(* Logix 5000 project; controller SX_V040001_C001 vendor 1 type 14 code 77 rev 16.23; software revision 16.04; part 12 of 35 *)
(* tags used below, declared in another part *)
   ALL_KINDS : INT[90];
   Basic : INT;
   C_MINUTES : COUNTER;
   C_SECONDS : COUNTER;
   CMD : INT[36];
   DRIVE : INT[32];
   DRIVE_INTERVAL : INT[8];
   EMPTYING : INT[18];
   G_DInput : DINT[3];
   G_DOutput : DINT[3];
   loading : INT[19];
   louvre : INT[11];
   m_alarm_exist : BOOL;
   m_alarm_horn : BOOL;
   m_battery_low : BOOL;
   m_on_off_line : BOOL;
   m_power_up : BOOL;
   PARAMETER : INT[501];
   STATUS_GENERAL : INT[135];
   TEMP : INT[14];
(* MainProgram, continued *)

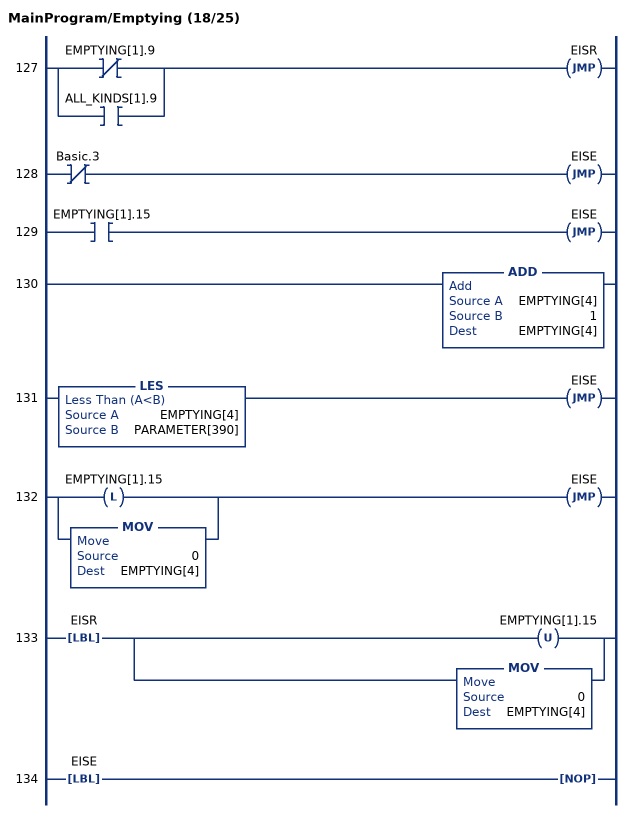
   [picture p256: MainProgram/Emptying rungs 127-134]
   127: [XIO(EMPTYING[1].9) ,XIC(ALL_KINDS[1].9) ]JMP(EISR);
   128: XIO(Basic.3)JMP(EISE);
   129: XIC(EMPTYING[1].15)JMP(EISE);
   130: ADD(EMPTYING[4],1,EMPTYING[4]);
   131: LES(EMPTYING[4],PARAMETER[390])JMP(EISE);
   132: [OTL(EMPTYING[1].15) ,MOV(0,EMPTYING[4]) ]JMP(EISE);
   133: LBL(EISR)[OTU(EMPTYING[1].15) ,MOV(0,EMPTYING[4]) ];
   134: LBL(EISE)NOP();
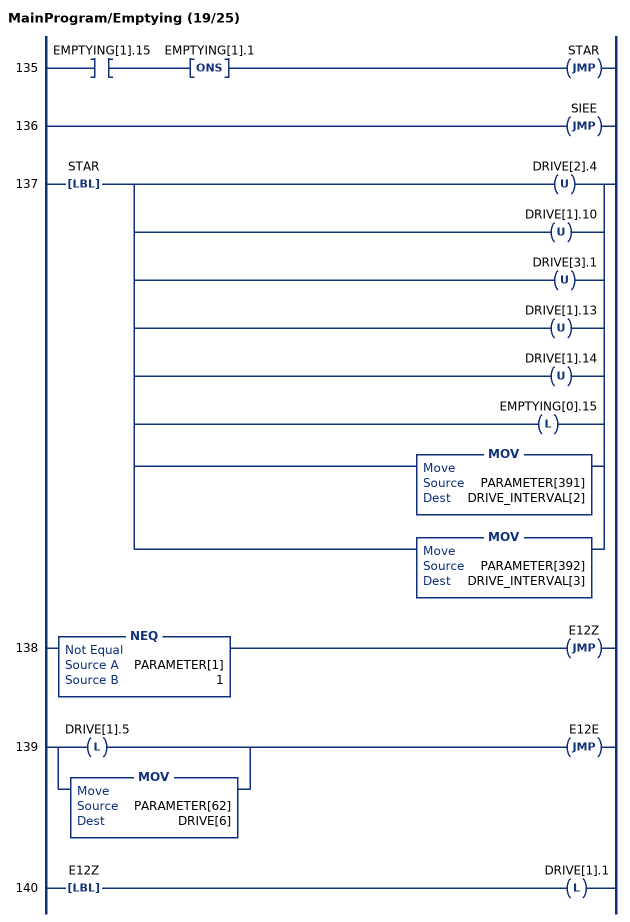
   135: XIC(EMPTYING[1].15)ONS(EMPTYING[1].1)JMP(STAR);
   136: JMP(SIEE);
   137: LBL(STAR)[OTU(DRIVE[2].4) ,OTU(DRIVE[1].10) ,OTU(DRIVE[3].1) ,OTU(DRIVE[1].13) ,OTU(DRIVE[1].14) ,OTL(EMPTYING[0].15) ,MOV(PARAMETER[391],DRIVE_INTERVAL[2]) ,MOV(PARAMETER[392],DRIVE_INTERVAL[3]) ];
   138: NEQ(PARAMETER[1],1)JMP(E12Z);
   139: [OTL(DRIVE[1].5) ,MOV(PARAMETER[62],DRIVE[6]) ]JMP(E12E);
   140: LBL(E12Z)OTL(DRIVE[1].1);
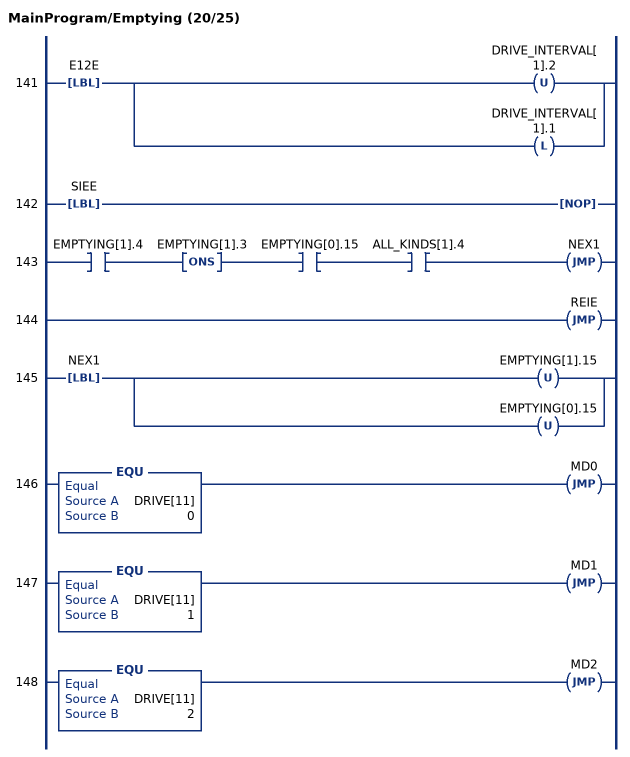
   141: LBL(E12E)[OTU(DRIVE_INTERVAL[1].2) ,OTL(DRIVE_INTERVAL[1].1) ];
   142: LBL(SIEE)NOP();
   143: XIC(EMPTYING[1].4)ONS(EMPTYING[1].3)XIC(EMPTYING[0].15)XIC(ALL_KINDS[1].4)JMP(NEX1);
   144: JMP(REIE);
   145: LBL(NEX1)[OTU(EMPTYING[1].15) ,OTU(EMPTYING[0].15) ];
   146: EQU(DRIVE[11],0)JMP(MD0);
   147: EQU(DRIVE[11],1)JMP(MD1);
   148: EQU(DRIVE[11],2)JMP(MD2);
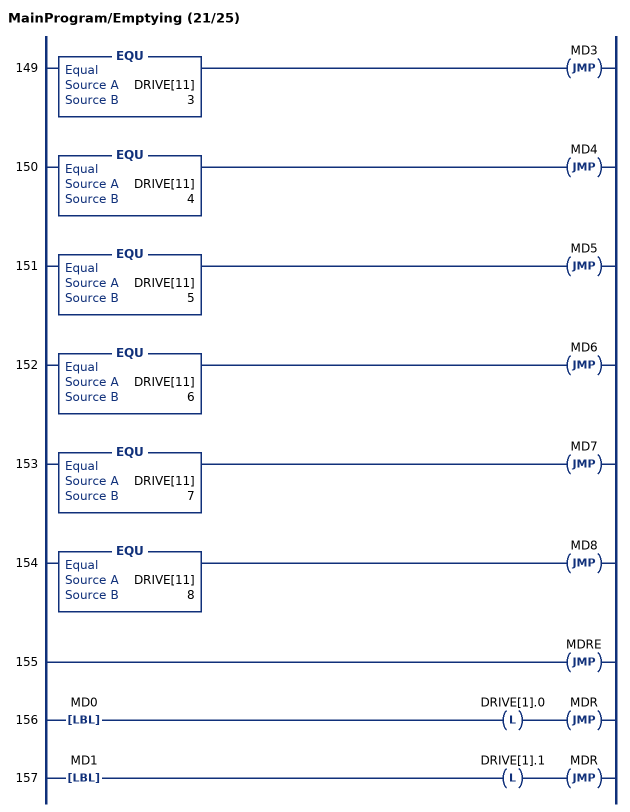
   149: EQU(DRIVE[11],3)JMP(MD3);
   150: EQU(DRIVE[11],4)JMP(MD4);
   151: EQU(DRIVE[11],5)JMP(MD5);
   152: EQU(DRIVE[11],6)JMP(MD6);
   153: EQU(DRIVE[11],7)JMP(MD7);
   154: EQU(DRIVE[11],8)JMP(MD8);
   155: JMP(MDRE);
   156: LBL(MD0)OTL(DRIVE[1].0)JMP(MDR);
   157: LBL(MD1)OTL(DRIVE[1].1)JMP(MDR);
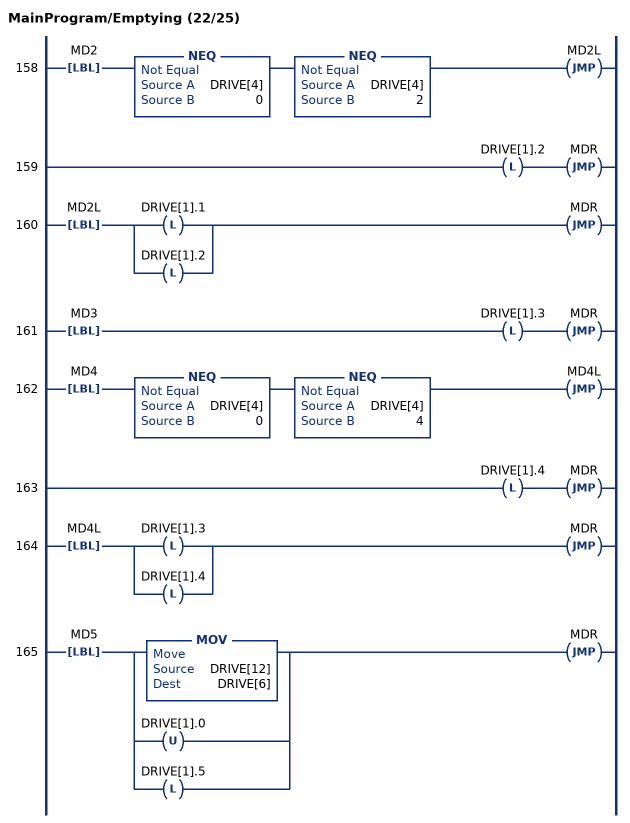
   158: LBL(MD2)NEQ(DRIVE[4],0)NEQ(DRIVE[4],2)JMP(MD2L);
   159: OTL(DRIVE[1].2)JMP(MDR);
   160: LBL(MD2L)[OTL(DRIVE[1].1) ,OTL(DRIVE[1].2) ]JMP(MDR);
   161: LBL(MD3)OTL(DRIVE[1].3)JMP(MDR);
   162: LBL(MD4)NEQ(DRIVE[4],0)NEQ(DRIVE[4],4)JMP(MD4L);
   163: OTL(DRIVE[1].4)JMP(MDR);
   164: LBL(MD4L)[OTL(DRIVE[1].3) ,OTL(DRIVE[1].4) ]JMP(MDR);
   165: LBL(MD5)[MOV(DRIVE[12],DRIVE[6]) ,OTU(DRIVE[1].0) ,OTL(DRIVE[1].5) ]JMP(MDR);
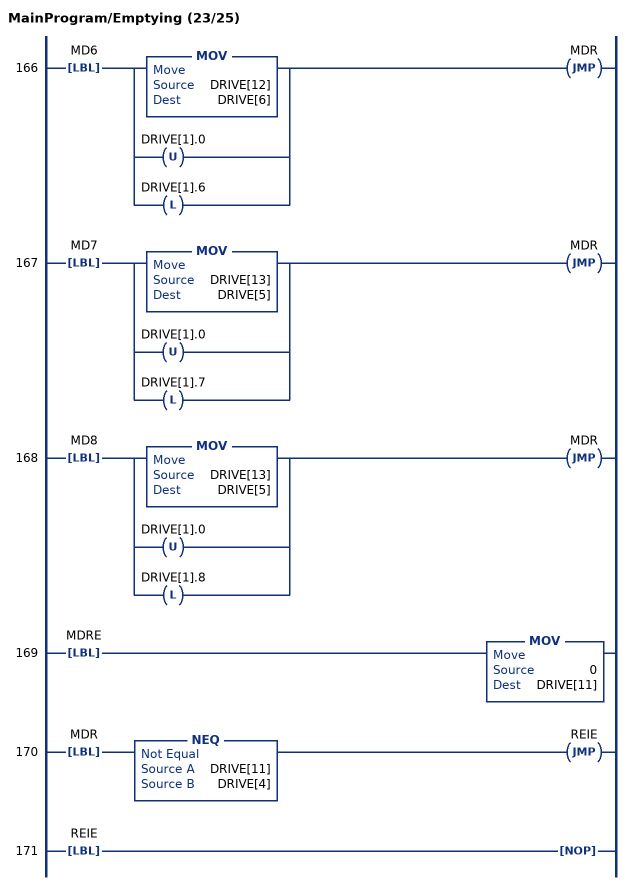
   166: LBL(MD6)[MOV(DRIVE[12],DRIVE[6]) ,OTU(DRIVE[1].0) ,OTL(DRIVE[1].6) ]JMP(MDR);
   167: LBL(MD7)[MOV(DRIVE[13],DRIVE[5]) ,OTU(DRIVE[1].0) ,OTL(DRIVE[1].7) ]JMP(MDR);
   168: LBL(MD8)[MOV(DRIVE[13],DRIVE[5]) ,OTU(DRIVE[1].0) ,OTL(DRIVE[1].8) ]JMP(MDR);
   169: LBL(MDRE)MOV(0,DRIVE[11]);
   170: LBL(MDR)NEQ(DRIVE[11],DRIVE[4])JMP(REIE);
   171: LBL(REIE)NOP();
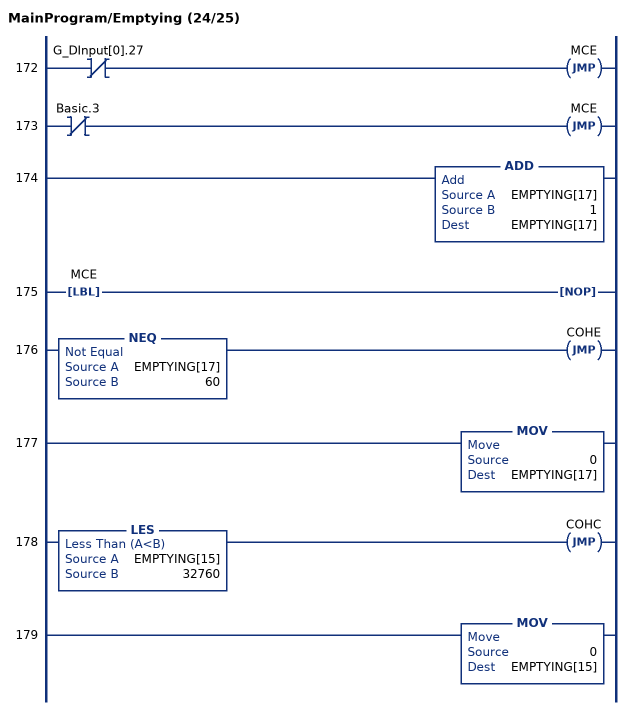
   172: XIO(G_DInput[0].27)JMP(MCE);
   173: XIO(Basic.3)JMP(MCE);
   174: ADD(EMPTYING[17],1,EMPTYING[17]);
   175: LBL(MCE)NOP();
   176: NEQ(EMPTYING[17],60)JMP(COHE);
   177: MOV(0,EMPTYING[17]);
   178: LES(EMPTYING[15],32760)JMP(COHC);
   179: MOV(0,EMPTYING[15]);
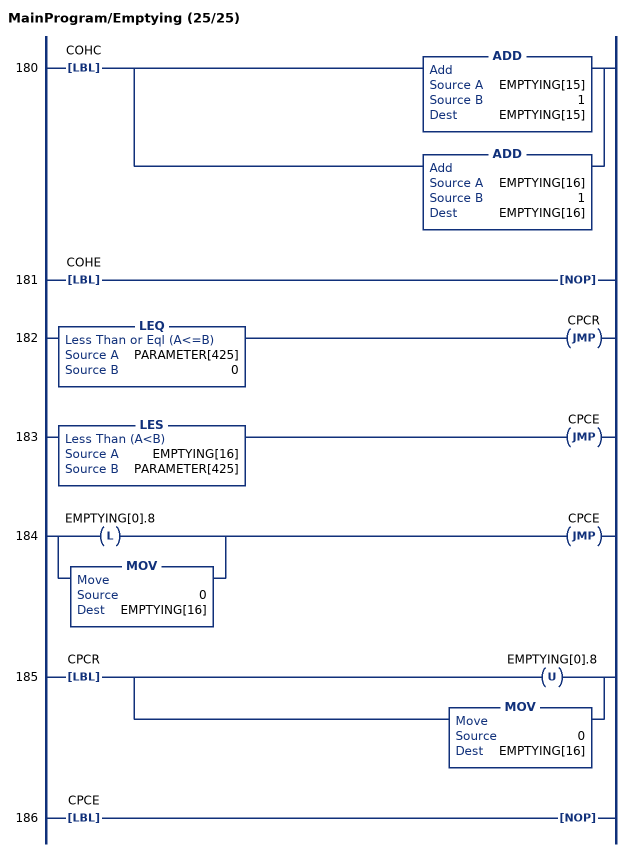
   180: LBL(COHC)[ADD(EMPTYING[15],1,EMPTYING[15]) ,ADD(EMPTYING[16],1,EMPTYING[16]) ];
   181: LBL(COHE)NOP();
   182: LEQ(PARAMETER[425],0)JMP(CPCR);
   183: LES(EMPTYING[16],PARAMETER[425])JMP(CPCE);
   184: [OTL(EMPTYING[0].8) ,MOV(0,EMPTYING[16]) ]JMP(CPCE);
   185: LBL(CPCR)[OTU(EMPTYING[0].8) ,MOV(0,EMPTYING[16]) ];
   186: LBL(CPCE)NOP();
END_ROUTINE

ROUTINE FirstScan   (* ladder *)
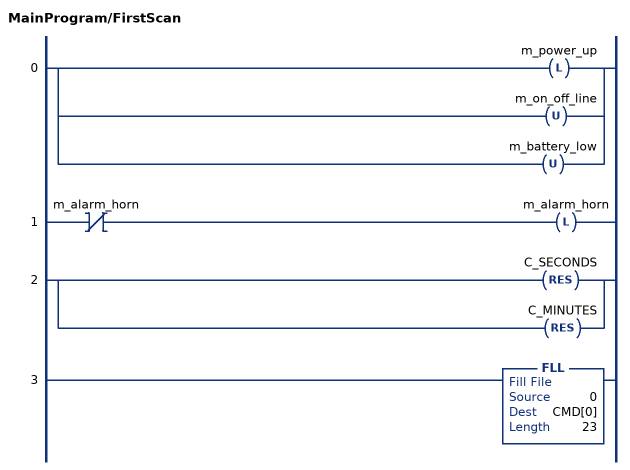
   0: [OTL(m_power_up) ,OTU(m_on_off_line) ,OTU(m_battery_low) ];
   1: XIO(m_alarm_horn)OTL(m_alarm_horn);
   2: [RES(C_SECONDS) ,RES(C_MINUTES) ];
   3: FLL(0,CMD[0],23);
END_ROUTINE

ROUTINE GenerateStatus   (* ladder *)
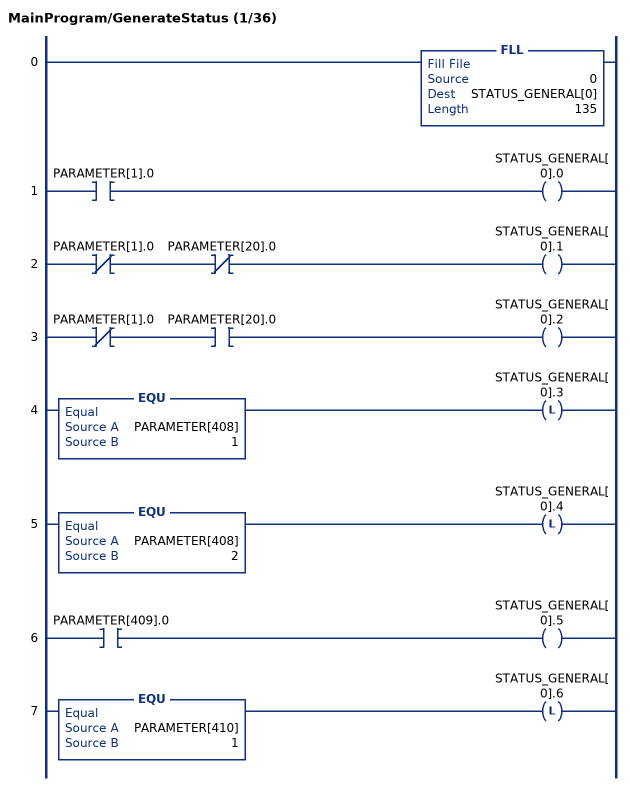
   0: FLL(0,STATUS_GENERAL[0],135);
   1: XIC(PARAMETER[1].0)OTE(STATUS_GENERAL[0].0);
   2: XIO(PARAMETER[1].0)XIO(PARAMETER[20].0)OTE(STATUS_GENERAL[0].1);
   3: XIO(PARAMETER[1].0)XIC(PARAMETER[20].0)OTE(STATUS_GENERAL[0].2);
   4: EQU(PARAMETER[408],1)OTL(STATUS_GENERAL[0].3);
   5: EQU(PARAMETER[408],2)OTL(STATUS_GENERAL[0].4);
   6: XIC(PARAMETER[409].0)OTE(STATUS_GENERAL[0].5);
   7: EQU(PARAMETER[410],1)OTL(STATUS_GENERAL[0].6);
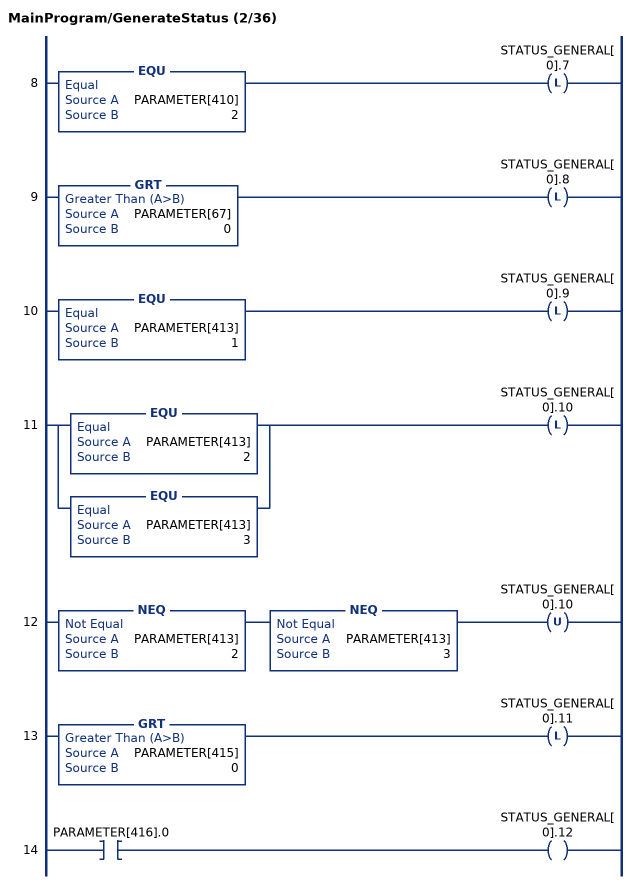
   8: EQU(PARAMETER[410],2)OTL(STATUS_GENERAL[0].7);
   9: GRT(PARAMETER[67],0)OTL(STATUS_GENERAL[0].8);
   10: EQU(PARAMETER[413],1)OTL(STATUS_GENERAL[0].9);
   11: [EQU(PARAMETER[413],2) ,EQU(PARAMETER[413],3) ]OTL(STATUS_GENERAL[0].10);
   12: NEQ(PARAMETER[413],2)NEQ(PARAMETER[413],3)OTU(STATUS_GENERAL[0].10);
   13: GRT(PARAMETER[415],0)OTL(STATUS_GENERAL[0].11);
   14: XIC(PARAMETER[416].0)OTE(STATUS_GENERAL[0].12);
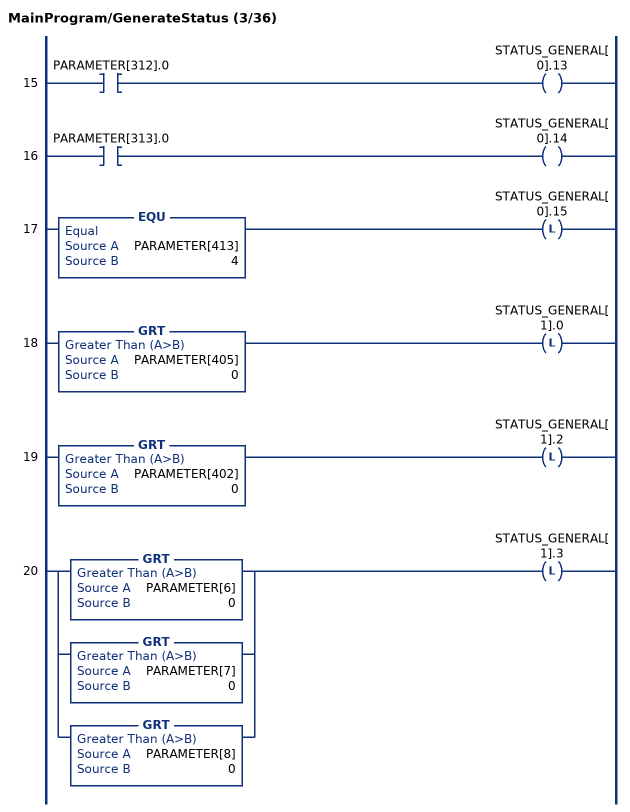
   15: XIC(PARAMETER[312].0)OTE(STATUS_GENERAL[0].13);
   16: XIC(PARAMETER[313].0)OTE(STATUS_GENERAL[0].14);
   17: EQU(PARAMETER[413],4)OTL(STATUS_GENERAL[0].15);
   18: GRT(PARAMETER[405],0)OTL(STATUS_GENERAL[1].0);
   19: GRT(PARAMETER[402],0)OTL(STATUS_GENERAL[1].2);
   20: [GRT(PARAMETER[6],0) ,GRT(PARAMETER[7],0) ,GRT(PARAMETER[8],0) ]OTL(STATUS_GENERAL[1].3);
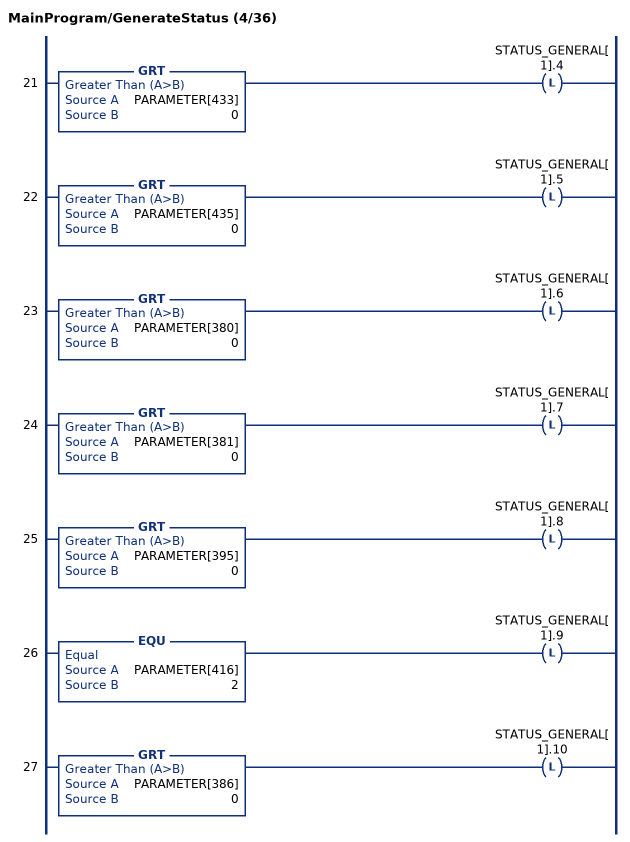
   21: GRT(PARAMETER[433],0)OTL(STATUS_GENERAL[1].4);
   22: GRT(PARAMETER[435],0)OTL(STATUS_GENERAL[1].5);
   23: GRT(PARAMETER[380],0)OTL(STATUS_GENERAL[1].6);
   24: GRT(PARAMETER[381],0)OTL(STATUS_GENERAL[1].7);
   25: GRT(PARAMETER[395],0)OTL(STATUS_GENERAL[1].8);
   26: EQU(PARAMETER[416],2)OTL(STATUS_GENERAL[1].9);
   27: GRT(PARAMETER[386],0)OTL(STATUS_GENERAL[1].10);
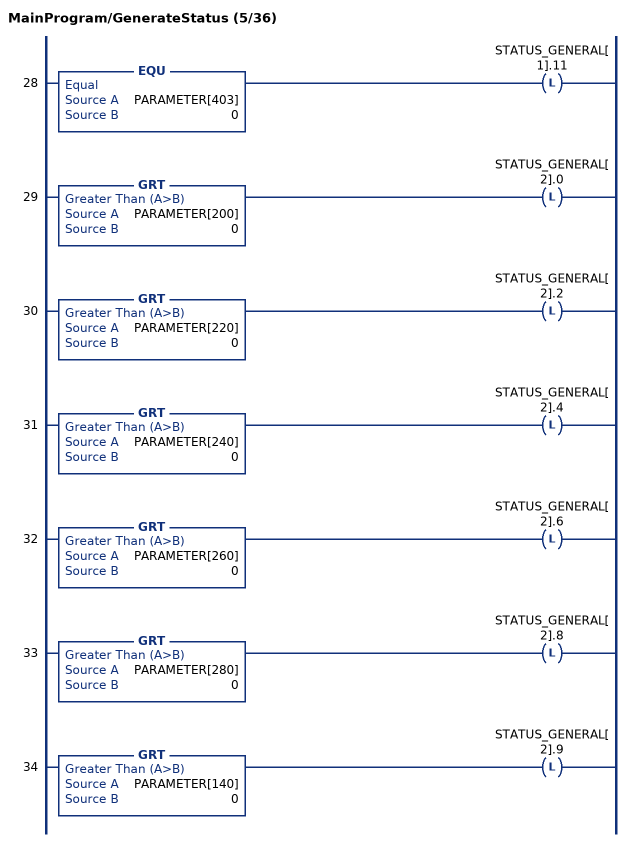
   28: EQU(PARAMETER[403],0)OTL(STATUS_GENERAL[1].11);
   29: GRT(PARAMETER[200],0)OTL(STATUS_GENERAL[2].0);
   30: GRT(PARAMETER[220],0)OTL(STATUS_GENERAL[2].2);
   31: GRT(PARAMETER[240],0)OTL(STATUS_GENERAL[2].4);
   32: GRT(PARAMETER[260],0)OTL(STATUS_GENERAL[2].6);
   33: GRT(PARAMETER[280],0)OTL(STATUS_GENERAL[2].8);
   34: GRT(PARAMETER[140],0)OTL(STATUS_GENERAL[2].9);
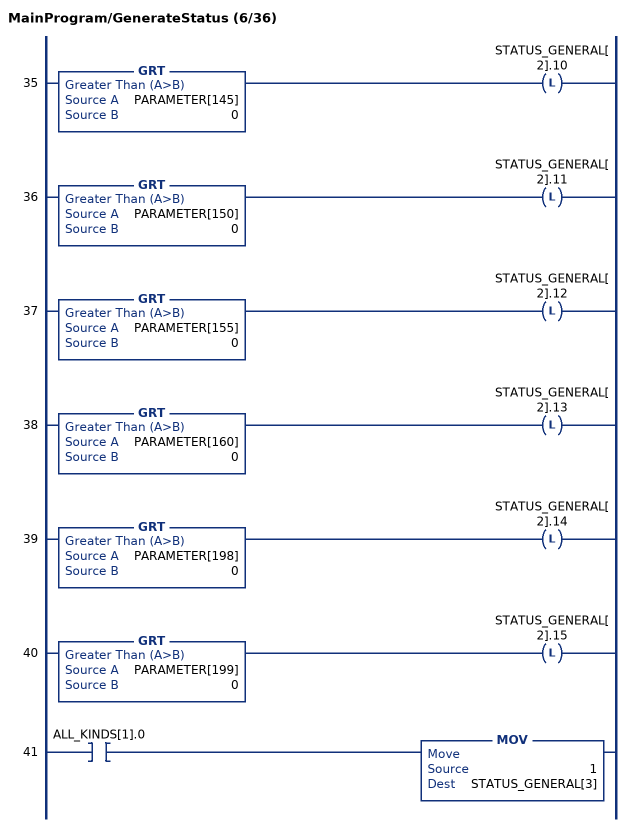
   35: GRT(PARAMETER[145],0)OTL(STATUS_GENERAL[2].10);
   36: GRT(PARAMETER[150],0)OTL(STATUS_GENERAL[2].11);
   37: GRT(PARAMETER[155],0)OTL(STATUS_GENERAL[2].12);
   38: GRT(PARAMETER[160],0)OTL(STATUS_GENERAL[2].13);
   39: GRT(PARAMETER[198],0)OTL(STATUS_GENERAL[2].14);
   40: GRT(PARAMETER[199],0)OTL(STATUS_GENERAL[2].15);
   41: XIC(ALL_KINDS[1].0)MOV(1,STATUS_GENERAL[3]);
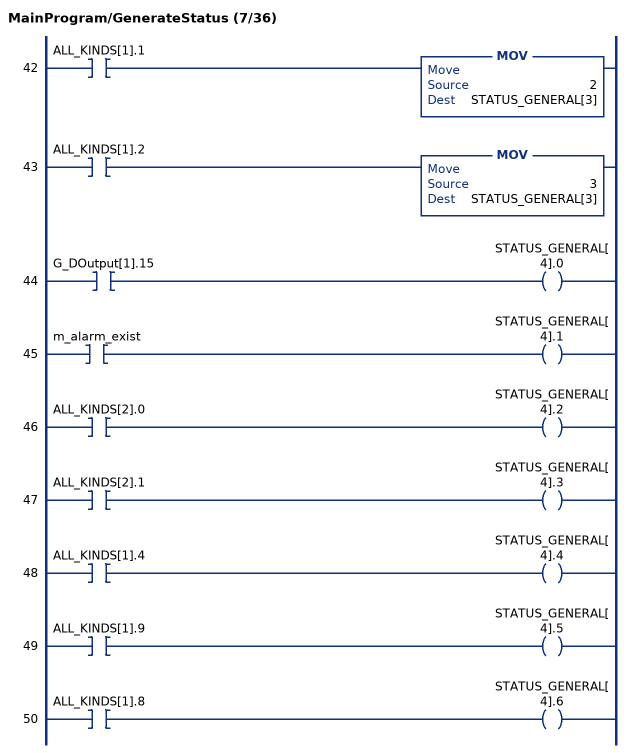
   42: XIC(ALL_KINDS[1].1)MOV(2,STATUS_GENERAL[3]);
   43: XIC(ALL_KINDS[1].2)MOV(3,STATUS_GENERAL[3]);
   44: XIC(G_DOutput[1].15)OTE(STATUS_GENERAL[4].0);
   45: XIC(m_alarm_exist)OTE(STATUS_GENERAL[4].1);
   46: XIC(ALL_KINDS[2].0)OTE(STATUS_GENERAL[4].2);
   47: XIC(ALL_KINDS[2].1)OTE(STATUS_GENERAL[4].3);
   48: XIC(ALL_KINDS[1].4)OTE(STATUS_GENERAL[4].4);
   49: XIC(ALL_KINDS[1].9)OTE(STATUS_GENERAL[4].5);
   50: XIC(ALL_KINDS[1].8)OTE(STATUS_GENERAL[4].6);
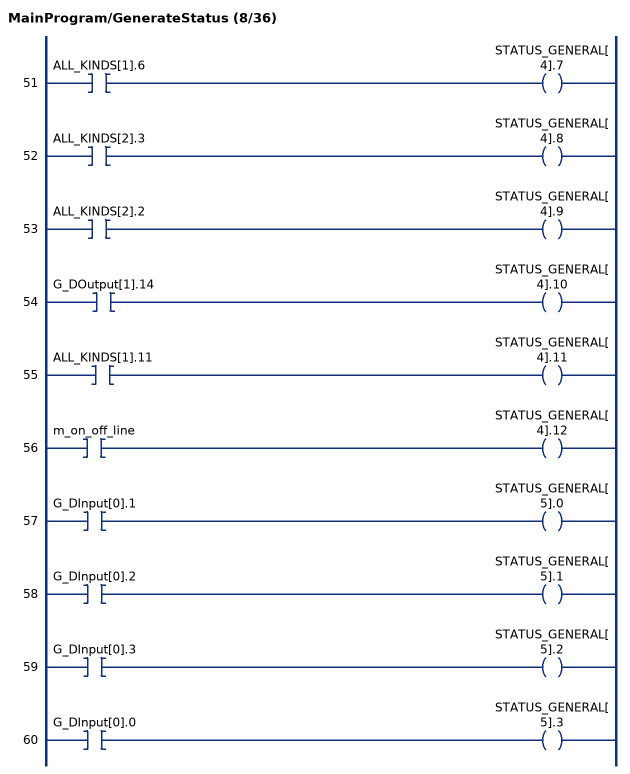
   51: XIC(ALL_KINDS[1].6)OTE(STATUS_GENERAL[4].7);
   52: XIC(ALL_KINDS[2].3)OTE(STATUS_GENERAL[4].8);
   53: XIC(ALL_KINDS[2].2)OTE(STATUS_GENERAL[4].9);
   54: XIC(G_DOutput[1].14)OTE(STATUS_GENERAL[4].10);
   55: XIC(ALL_KINDS[1].11)OTE(STATUS_GENERAL[4].11);
   56: XIC(m_on_off_line)OTE(STATUS_GENERAL[4].12);
   57: XIC(G_DInput[0].1)OTE(STATUS_GENERAL[5].0);
   58: XIC(G_DInput[0].2)OTE(STATUS_GENERAL[5].1);
   59: XIC(G_DInput[0].3)OTE(STATUS_GENERAL[5].2);
   60: XIC(G_DInput[0].0)OTE(STATUS_GENERAL[5].3);
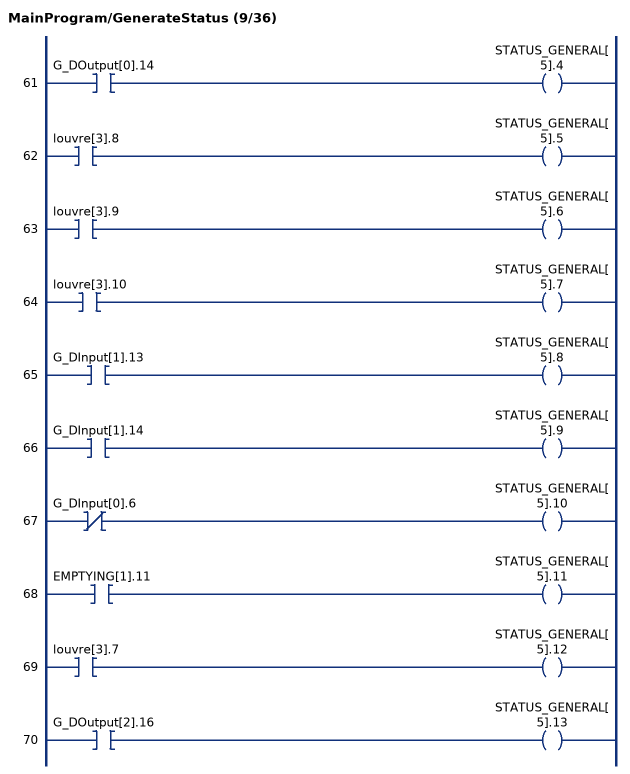
   61: XIC(G_DOutput[0].14)OTE(STATUS_GENERAL[5].4);
   62: XIC(louvre[3].8)OTE(STATUS_GENERAL[5].5);
   63: XIC(louvre[3].9)OTE(STATUS_GENERAL[5].6);
   64: XIC(louvre[3].10)OTE(STATUS_GENERAL[5].7);
   65: XIC(G_DInput[1].13)OTE(STATUS_GENERAL[5].8);
   66: XIC(G_DInput[1].14)OTE(STATUS_GENERAL[5].9);
   67: XIO(G_DInput[0].6)OTE(STATUS_GENERAL[5].10);
   68: XIC(EMPTYING[1].11)OTE(STATUS_GENERAL[5].11);
   69: XIC(louvre[3].7)OTE(STATUS_GENERAL[5].12);
   70: XIC(G_DOutput[2].16)OTE(STATUS_GENERAL[5].13);
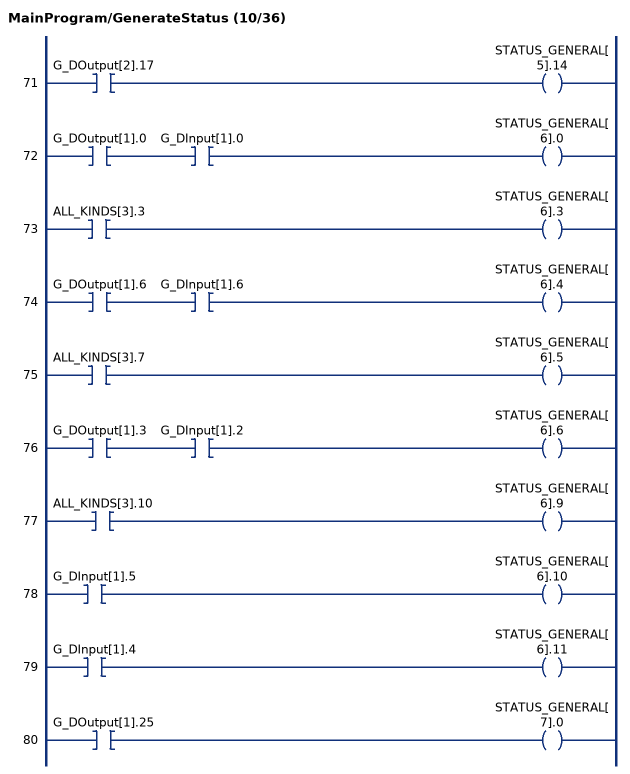
   71: XIC(G_DOutput[2].17)OTE(STATUS_GENERAL[5].14);
   72: XIC(G_DOutput[1].0)XIC(G_DInput[1].0)OTE(STATUS_GENERAL[6].0);
   73: XIC(ALL_KINDS[3].3)OTE(STATUS_GENERAL[6].3);
   74: XIC(G_DOutput[1].6)XIC(G_DInput[1].6)OTE(STATUS_GENERAL[6].4);
   75: XIC(ALL_KINDS[3].7)OTE(STATUS_GENERAL[6].5);
   76: XIC(G_DOutput[1].3)XIC(G_DInput[1].2)OTE(STATUS_GENERAL[6].6);
   77: XIC(ALL_KINDS[3].10)OTE(STATUS_GENERAL[6].9);
   78: XIC(G_DInput[1].5)OTE(STATUS_GENERAL[6].10);
   79: XIC(G_DInput[1].4)OTE(STATUS_GENERAL[6].11);
   80: XIC(G_DOutput[1].25)OTE(STATUS_GENERAL[7].0);
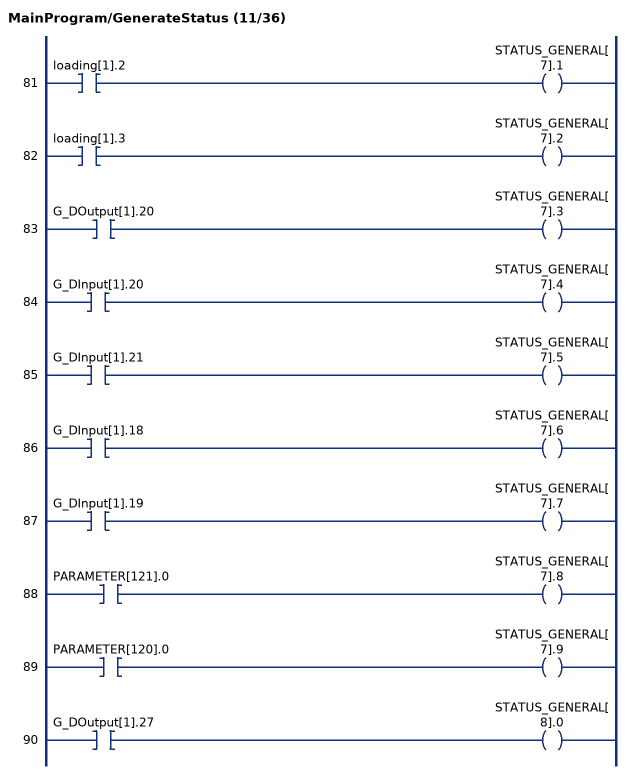
   81: XIC(loading[1].2)OTE(STATUS_GENERAL[7].1);
   82: XIC(loading[1].3)OTE(STATUS_GENERAL[7].2);
   83: XIC(G_DOutput[1].20)OTE(STATUS_GENERAL[7].3);
   84: XIC(G_DInput[1].20)OTE(STATUS_GENERAL[7].4);
   85: XIC(G_DInput[1].21)OTE(STATUS_GENERAL[7].5);
   86: XIC(G_DInput[1].18)OTE(STATUS_GENERAL[7].6);
   87: XIC(G_DInput[1].19)OTE(STATUS_GENERAL[7].7);
   88: XIC(PARAMETER[121].0)OTE(STATUS_GENERAL[7].8);
   89: XIC(PARAMETER[120].0)OTE(STATUS_GENERAL[7].9);
   90: XIC(G_DOutput[1].27)OTE(STATUS_GENERAL[8].0);
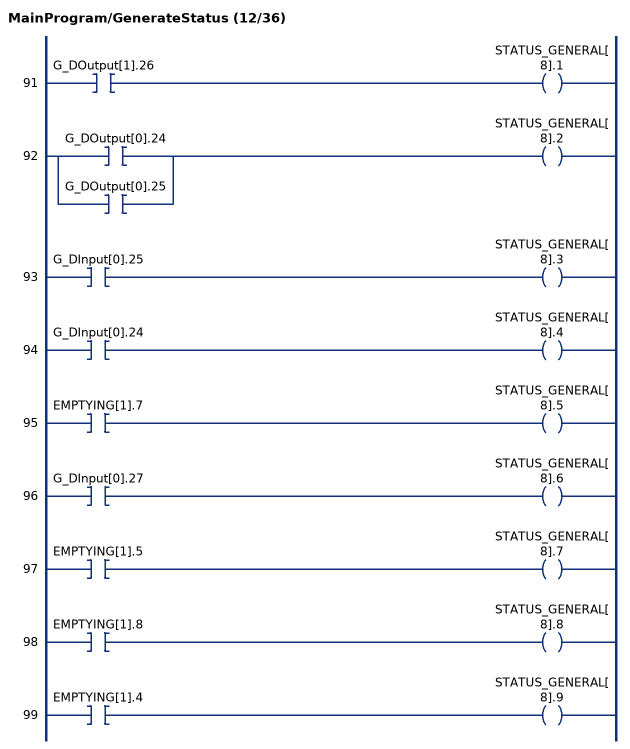
   91: XIC(G_DOutput[1].26)OTE(STATUS_GENERAL[8].1);
   92: [XIC(G_DOutput[0].24) ,XIC(G_DOutput[0].25) ]OTE(STATUS_GENERAL[8].2);
   93: XIC(G_DInput[0].25)OTE(STATUS_GENERAL[8].3);
   94: XIC(G_DInput[0].24)OTE(STATUS_GENERAL[8].4);
   95: XIC(EMPTYING[1].7)OTE(STATUS_GENERAL[8].5);
   96: XIC(G_DInput[0].27)OTE(STATUS_GENERAL[8].6);
   97: XIC(EMPTYING[1].5)OTE(STATUS_GENERAL[8].7);
   98: XIC(EMPTYING[1].8)OTE(STATUS_GENERAL[8].8);
   99: XIC(EMPTYING[1].4)OTE(STATUS_GENERAL[8].9);
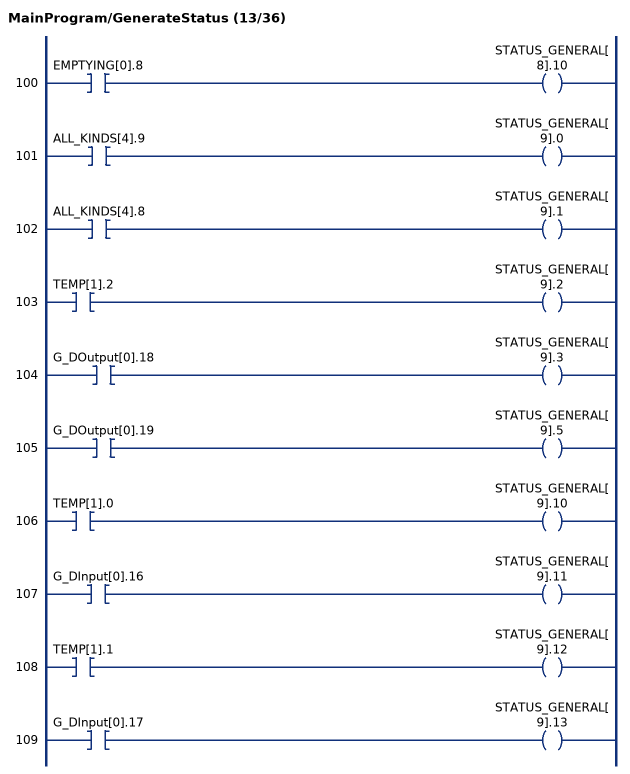
   100: XIC(EMPTYING[0].8)OTE(STATUS_GENERAL[8].10);
   101: XIC(ALL_KINDS[4].9)OTE(STATUS_GENERAL[9].0);
   102: XIC(ALL_KINDS[4].8)OTE(STATUS_GENERAL[9].1);
   103: XIC(TEMP[1].2)OTE(STATUS_GENERAL[9].2);
   104: XIC(G_DOutput[0].18)OTE(STATUS_GENERAL[9].3);
   105: XIC(G_DOutput[0].19)OTE(STATUS_GENERAL[9].5);
   106: XIC(TEMP[1].0)OTE(STATUS_GENERAL[9].10);
   107: XIC(G_DInput[0].16)OTE(STATUS_GENERAL[9].11);
   108: XIC(TEMP[1].1)OTE(STATUS_GENERAL[9].12);
   109: XIC(G_DInput[0].17)OTE(STATUS_GENERAL[9].13);
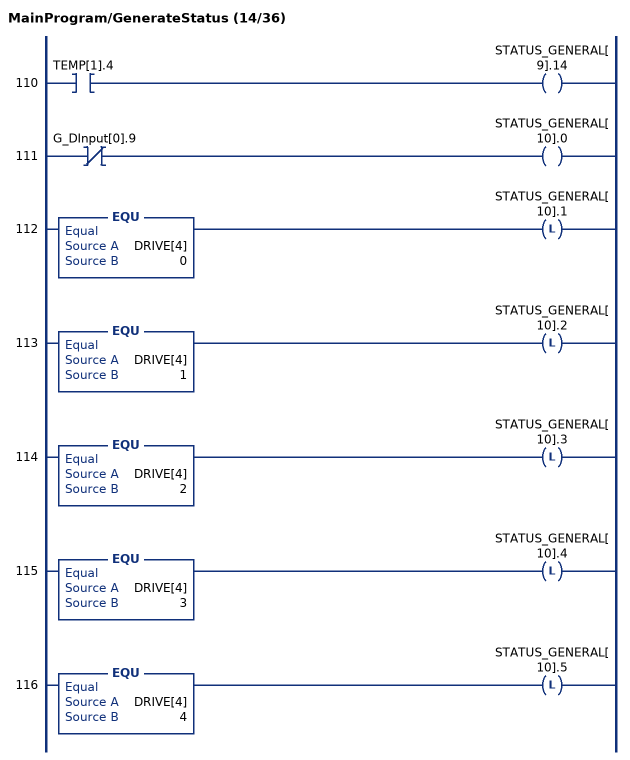
   110: XIC(TEMP[1].4)OTE(STATUS_GENERAL[9].14);
   111: XIO(G_DInput[0].9)OTE(STATUS_GENERAL[10].0);
   112: EQU(DRIVE[4],0)OTL(STATUS_GENERAL[10].1);
   113: EQU(DRIVE[4],1)OTL(STATUS_GENERAL[10].2);
   114: EQU(DRIVE[4],2)OTL(STATUS_GENERAL[10].3);
   115: EQU(DRIVE[4],3)OTL(STATUS_GENERAL[10].4);
   116: EQU(DRIVE[4],4)OTL(STATUS_GENERAL[10].5);
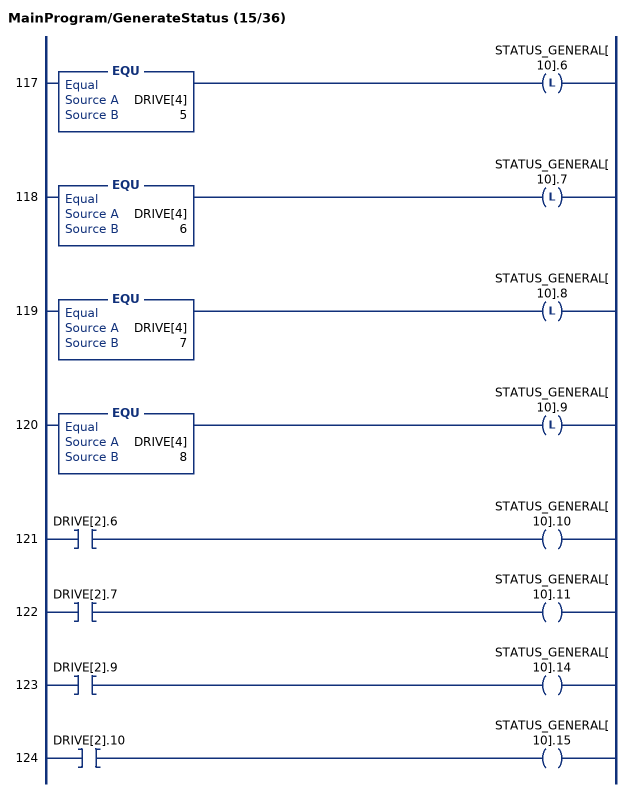
   117: EQU(DRIVE[4],5)OTL(STATUS_GENERAL[10].6);
   118: EQU(DRIVE[4],6)OTL(STATUS_GENERAL[10].7);
   119: EQU(DRIVE[4],7)OTL(STATUS_GENERAL[10].8);
   120: EQU(DRIVE[4],8)OTL(STATUS_GENERAL[10].9);
   121: XIC(DRIVE[2].6)OTE(STATUS_GENERAL[10].10);
   122: XIC(DRIVE[2].7)OTE(STATUS_GENERAL[10].11);
   123: XIC(DRIVE[2].9)OTE(STATUS_GENERAL[10].14);
   124: XIC(DRIVE[2].10)OTE(STATUS_GENERAL[10].15);
